TYPE T_Ctrl_SIf_PTS_Out :
STRUCT
END_STRUCT
END_TYPE

(* stored: Version 1.1.0.1, ProductVersion 3.1.0.19
   DUT T_Ctrl_SIf_PTS_Out: Id {23ef33b4-c1f0-4093-8901-5116478a0b44} *)
